    FOR _eInst := E_INSTANCE.BUFFER_INFEED TO E_INSTANCE.SENDER_BUFFER_INFEED
    DO
      // handshakes to instances: 
      // - deconstruct this for your own implementation
      CASE _InstanceState[_eInst].State
      OF
        E_INSTANCE_STATE.DISABLED:
          CASE _InstanceState[_eInst].Progress
          OF
            E_PROGRESS.PROGRESS_BUSY:
              _InstanceCtrl[_eInst].Cmd    := E_INSTANCE_CMD.ENABLE;
          END_CASE
      
        E_INSTANCE_STATE.ENABLED:
          CASE _InstanceState[_eInst].Progress
          OF
            E_PROGRESS.PROGRESS_OCCUPIED:
              _InstanceCtrl[_eInst].Cmd    := E_INSTANCE_CMD.PROCEED;
          END_CASE

        E_INSTANCE_STATE.WORKING:
          CASE _InstanceState[_eInst].Progress
          OF
            E_PROGRESS.PROGRESS_BUSY:
              _tonProcess [_eInst]
                              (IN         := FALSE, 
                               PT         := _tProcess[_eInst]);


              IF (_eInst > E_INSTANCE.OUTFEED_ROBOT_R2) OR
                 (_eInst < E_INSTANCE.OUTFEED_ROBOT_R1) OR
                 (_bSingleOutput) OR
                 NOT (GVL_APPLICATION.bOutput_R1R2)
              THEN
                _InstanceCtrl[_eInst].Cmd   := E_INSTANCE_CMD.WORK;
              ELSE
                IF (_InstanceState[E_INSTANCE.OUTFEED_ROBOT_R1].State = 
                    _InstanceState[E_INSTANCE.OUTFEED_ROBOT_R2].State )
                THEN
                  // in this example the outfeed instances are working in sync
                  _InstanceCtrl[_eInst].Cmd := E_INSTANCE_CMD.WORK;
                END_IF
              END_IF
      
      
            E_PROGRESS.PROGRESS_CHECK:
              _tonProcess [_eInst]
                              (IN         := TRUE, 
                               PT         := _tProcess[_eInst]);
      
              IF _tonProcess [_eInst].Q
              THEN
                _InstanceCtrl[_eInst].Cmd := E_INSTANCE_CMD.FINISH;
              END_IF
          END_CASE


        E_INSTANCE_STATE.FINISH:
          CASE _InstanceState[_eInst].Progress
          OF
            E_PROGRESS.PROGRESS_BUSY:
              _tonProcess [_eInst]
                              (IN         := FALSE, 
                               PT         := _tProcess[_eInst]);

              _InstanceCtrl[_eInst].Cmd    := E_INSTANCE_CMD.FINISH;

            E_PROGRESS.PROGRESS_OCCUPIED:
              _InstanceCtrl[_eInst].Cmd    := E_INSTANCE_CMD.PROCEED;
          END_CASE
        END_CASE
    END_FOR
END_CASE
//-----------------------------------------------------------------------------
//-----------------------------------------------------------------------------

Work                            := _eState;
END_METHOD

PROPERTY WriteTimeVariant : bool
GET
WriteTimeVariant := _bWriteTimeVariant;
END_GET
SET
_bWriteTimeVariant := WriteTimeVariant;
END_SET
END_PROPERTY

PROPERTY XtsTransportCtrl : REFERENCE TO ST_XTS_TRANSPORT_CTRL
SET
_XtsTransportCtrl REF= XtsTransportCtrl;
END_SET
END_PROPERTY

PROPERTY XtsTransportState : REFERENCE TO ST_XTS_TRANSPORT_STATE
SET
_XtsTransportState REF= XtsTransportState;
END_SET
END_PROPERTY

END_FUNCTION_BLOCK

(* stored: Version 1.1.0.1, ProductVersion 3.1.4026.13
   POU fb_Application: Id {2a567699-b424-4e74-9f05-5574e5bc55b4}, SpecialFunc None
   Folder methods: Id {c1859e40-d269-4bfd-b7e9-641110aadb02}
   Folder properties: Id {440d7726-2a35-48b4-b212-3894cea03b12}
   Method Check: Id {b52b527b-139a-44b4-ab60-3e8b71488a0f}
   Method Clear: Id {a3ccc2ba-024d-44f1-adda-ac1f1be496a7}
   Method Cmd: Id {5496702b-60b7-475b-bef7-df563de1292d}
   Property CollectorInterface: Id {098e7272-6200-4a40-80ef-8c196e915eab}
   Set Set: Id {895034ec-84e5-4403-8b5f-9feedb87d7e4}
   Property Ctrl: Id {046d33ef-169b-4a2a-8c66-b97cf29ea596}
   Set Set: Id {a97b0d64-fc43-43a2-a267-33d710f4a902}
   Method Disable: Id {f3dd121e-604a-495b-ae98-29c9fcd2c0d9}
   Method Enable: Id {7ca4f60a-d1e0-4397-a83a-ed8dcb1017aa}
   Method Finish: Id {5b10ef5d-aac9-4514-b56a-99e09c68d7d2}
   Method Init: Id {10e2e475-1124-4c32-9d48-21872f6d1b74}
   Property InstanceCtrl: Id {7acdd1cc-198f-40bb-ba40-7856faf0d91c}
   Set Set: Id {2d3d313b-7311-479e-b918-28346a8bce77}
   Property InstanceState: Id {c2466ee2-4a57-4083-9c87-9e9f7eba2a74}
   Set Set: Id {e5a17682-314e-4e49-9b97-297ce85960e3}
   Method ListData: Id {8b730337-4e4b-4900-b4e8-13a7fa236b19}
   Property MessageLevel: Id {8ade6450-90c5-4683-b47c-6063ab1cfae3}
   Get Get: Id {b8718ada-c11b-4f81-b30a-3da434a9b4eb}
   Set Set: Id {16f6be41-bbda-46b4-a576-479cb4060503}
   Method Proceed: Id {f9a2f6e2-08f8-408b-a37e-4b3a16a77892}
   Property ProcessLinkedLists: Id {841e2785-8a81-4dab-ab69-a2404506471d}
   Set Set: Id {df60a9ec-7446-4a8a-92e2-3d5f72426dde}
   Property State: Id {257b9e36-771d-4714-8e16-430670e6fe24}
   Set Set: Id {588232c9-69de-48cc-813f-9f958d7bf6a6}
   Method Work: Id {c9245136-972a-4403-803b-e5d1ec9271e9}
   Property WriteTimeVariant: Id {741bcc54-9ee2-4811-8354-d070bf4ab52f}
   Get Get: Id {10a241a2-b4c9-46fa-b817-d2141a3ed1bb}
   Set Set: Id {a4dacca1-c32a-41f0-a14c-c44274b906db}
   Property XtsTransportCtrl: Id {3391bec1-98d1-4039-b0cc-fd4068165ffc}
   Set Set: Id {4fe1f55c-1a91-41e0-ad15-d1076bfbadce}
   Property XtsTransportState: Id {fa356716-e420-4889-891d-40c9f915f287}
   Set Set: Id {caa6f3cc-431a-488e-b079-3523f2bff879} *)
